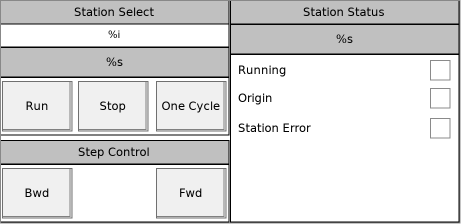
VISUALIZATION MANUAL_STEP  // 461x224
    Rectangle (0,22 229x25), "%i", text variable: Global_Variables_HMI.T_Curr_Step_Station, input disabled if: Global_Variables.M_StepRun
        OnMouseDown: write the text variable via VisuDialogs.Numpad, min 2, max 8
    Rectangle (0,47 229x30), "%s", text variable: Global_Variables_HMI.V_StepRunCurrStation
    Rectangle (0,0 229x24)
    RoundedRectangle (20,-3 188x30), "Station Select"
    Rectangle (0,77 229x58)
    Button (2,81 70x50), "Run"
        tap Global_Variables_HMI.T_StepRun
    Button (78,81 70x50), "Stop"
        tap Global_Variables_HMI.T_StepStop
    Button (156,81 70x50), "One Cycle", pressed state: Global_Variables_HMI.T_OneCycleRun
        toggle Global_Variables_HMI.T_OneCycleRun
    Rectangle (0,140 229x24)
    RoundedRectangle (20,137 188x30), "Step Control"
    Rectangle (0,164 229x58)
    Button (2,168 70x50), "Bwd"
        tap Global_Variables_HMI.T_StepBwd
    Button (156,168 70x50), "Fwd"
        tap Global_Variables_HMI.T_StepFwd
    Rectangle (230,0 229x24)
    RoundedRectangle (250,-3 188x30), "Station Status"
    Rectangle (230,54 229x168)
    RoundedRectangle (235,55 95x30), "Running"
    RoundedRectangle (235,83 95x30), "Origin"
    RoundedRectangle (235,113 95x30), "Station Error"
    Rectangle (230,24 229x30), "%s", text variable: Global_Variables_HMI.V_StepRunStatus
    Frame (430,118 20x20)
        shows Red_Ind(m_Input_Inst := Global_Variables_HMI.T_StationError)
    Frame (430,88 20x20)
        shows Green_Ind(m_Input_Inst := Global_Variables_HMI.T_Origin)
    Frame (430,60 20x20)
        shows Green_Ind(m_Input_Inst := Global_Variables.M_StepRun)
END_VISUALIZATION

(* stored: Version 1.1.0.1, ProductVersion 3.1.4018.2
   Visu MANUAL_STEP: Id {f2f97757-0b87-48e1-9c2f-d438a6f09ff0} *)
